SUBAPPLICATION HandshakePatternDemoIO (* Handshake pattern demo wired to physical I/O: a button (logiBUS_IE) triggers the Requester, an LED (logiBUS_QX) toggles once the handshake round-trip (REQ->CNF) has completed *)
  (* Standard: 61499-2; Description: Copyright (c) 2026 Meisterschulen am Ostbahnhof This program and the accompanying materials are made available under the terms of the Eclipse Public License 2.0 which is available at https://www.eclipse.org/legal/epl-2.0/ SPDX-License-Identifier: EPL-2.0 *)
  (* Version 1.0, 2026-08-31, Franz Höpfinger, Meisterschulen am Ostbahnhof, Handshake design pattern (IEC 61499 primer course, Module 6, Valeriy Vyatkin), physical I/O wrapper around HandshakePatternDemo - button/LED wiring style taken from test_B/Uebungen/Uebung_004a.SUB *)
  PACKAGE Meins::DesingPatterns::HandshakePattern;
  IMPORT logiBUS::io::DI::logiBUS_DI::Input_I1;
  IMPORT logiBUS::io::DI::logiBUS_DI_Events::BUTTON_SINGLE_CLICK;
  IMPORT logiBUS::io::DQ::logiBUS_DO::Output_Q1;
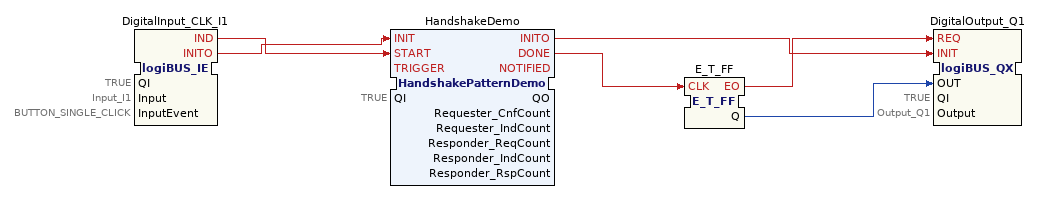
  FBS
    DigitalInput_CLK_I1 : logiBUS::io::DI::logiBUS_IE(QI := TRUE, Input := Input_I1, InputEvent := BUTTON_SINGLE_CLICK);
    E_T_FF : iec61499::events::E_T_FF;
    DigitalOutput_Q1 : logiBUS::io::DQ::logiBUS_QX(QI := TRUE, Output := Output_Q1);
  END_FBS
  SUBAPPS
    HandshakeDemo : Meins::DesingPatterns::HandshakePattern::HandshakePatternDemo(QI := TRUE);
  END_SUBAPPS
  EVENT_CONNECTIONS
    DigitalInput_CLK_I1.IND TO HandshakeDemo.START; (* Button press starts the handshake: the Requester sends REQ *)
    HandshakeDemo.DONE TO E_T_FF.CLK; (* Toggle the LED only once the Responder's CNF actually came back *)
    E_T_FF.EO TO DigitalOutput_Q1.REQ;
    DigitalInput_CLK_I1.INITO TO HandshakeDemo.INIT;
    HandshakeDemo.INITO TO DigitalOutput_Q1.INIT;
  END_CONNECTIONS
  DATA_CONNECTIONS
    E_T_FF.Q TO DigitalOutput_Q1.OUT;
  END_CONNECTIONS
END_SUBAPPLICATION
